TYPE ST_MachPar :
STRUCT
	InMoldDrying					: ST_IMDMachPar;
	ProductHandling					: ST_ProductHandlingMachPar;
END_STRUCT
END_TYPE

(* stored: Version 1.1.0.1, ProductVersion 3.1.4020.12
   DUT ST_MachPar: Id {cfb80fe3-ed42-4cbf-a7ca-fe26c95f2407} *)
